TYPE TProbingArea :
	(
		PA_BeforeSharpen := 0,
		PA_AfterSharpen,
		PA_WeightCalibration,
		PA_PartLayering1Offset0,
		PA_PartLayering1Offset1,
		PA_PartLayering2Offset0,
		PA_PartLayering2Offset1,
		PA_PartLayering3Offset0,
		PA_PartLayering3Offset1,
		PA_PartLayering4Offset0,
		PA_PartLayering4Offset1,
		PA_END
	);
END_TYPE

(* stored: Version 1.1.0.1, ProductVersion 3.1.4022.12
   DUT TProbingArea: Id {4acc44a2-0045-4e20-a22c-6b7b30ebb921} *)
